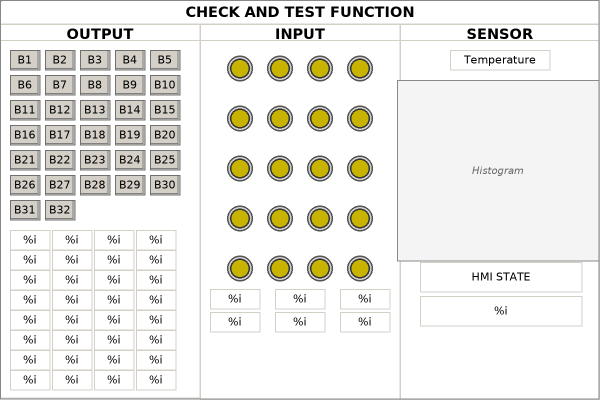
VISUALIZATION Set  // 600x400
    Textfield (0,0 600x24), "CHECK AND TEST FUNCTION"
    Rectangle (0,0 1x0)
    Textfield (0,24 200x20), "OUTPUT"
    Textfield (200,24 200x20), "INPUT"
    Textfield (400,24 200x20), "SENSOR"
    Textfield (0,40 200x358)
    Textfield (200,40 200x360)
    Textfield (400,40 200x360)
    Lamp1 (225,51 30x35), variable: HMI_Global.HMI_IN_Digital[0], style: Lamp-Lamp1-Yellow
    Lamp1 (265,51 30x35), variable: HMI_Global.HMI_IN_Digital[1], style: Lamp-Lamp1-Yellow
    Lamp1 (305,51 30x35), variable: HMI_Global.HMI_IN_Digital[2], style: Lamp-Lamp1-Yellow
    Lamp1 (345,51 30x35), variable: HMI_Global.HMI_IN_Digital[3], style: Lamp-Lamp1-Yellow
    Lamp1 (345,101 30x35), variable: HMI_Global.HMI_IN_Digital[7], style: Lamp-Lamp1-Yellow
    Lamp1 (225,101 30x35), variable: HMI_Global.HMI_IN_Digital[4], style: Lamp-Lamp1-Yellow
    Lamp1 (265,101 30x35), variable: HMI_Global.HMI_IN_Digital[5], style: Lamp-Lamp1-Yellow
    Lamp1 (305,101 30x35), variable: HMI_Global.HMI_IN_Digital[6], style: Lamp-Lamp1-Yellow
    Lamp1 (225,151 30x35), variable: HMI_Global.HMI_IN_Digital[8], style: Lamp-Lamp1-Yellow
    Lamp1 (345,151 30x35), variable: HMI_Global.HMI_IN_Digital[11], style: Lamp-Lamp1-Yellow
    Lamp1 (265,151 30x35), variable: HMI_Global.HMI_IN_Digital[9], style: Lamp-Lamp1-Yellow
    Lamp1 (305,151 30x35), variable: HMI_Global.HMI_IN_Digital[10], style: Lamp-Lamp1-Yellow
    Lamp1 (225,201 30x35), variable: HMI_Global.HMI_IN_Digital[12], style: Lamp-Lamp1-Yellow
    Lamp1 (265,201 30x35), variable: HMI_Global.HMI_IN_Digital[13], style: Lamp-Lamp1-Yellow
    Lamp1 (305,201 30x35), variable: HMI_Global.HMI_IN_Digital[14], style: Lamp-Lamp1-Yellow
    Lamp1 (345,201 30x35), variable: HMI_Global.HMI_IN_Digital[15], style: Lamp-Lamp1-Yellow
    Lamp1 (345,251 30x35), variable: HMI_Global.HMI_IN_Digital[20], style: Lamp-Lamp1-Yellow
    Lamp1 (225,251 30x35), variable: HMI_Global.HMI_IN_Digital[16], style: Lamp-Lamp1-Yellow
    Lamp1 (265,251 30x35), variable: HMI_Global.HMI_IN_Digital[17], style: Lamp-Lamp1-Yellow
    Lamp1 (305,251 30x35), variable: HMI_Global.HMI_IN_Digital[18], style: Lamp-Lamp1-Yellow
    Button (10,50 30x20), "B1"
        toggle HMI_Global.HMI_OUT_Digital[0]
    Textfield (210,289 50x20), "%i", text variable: HMI_Global.HMI_IN_Analog[0]
    Textfield (275,289 50x20), "%i", text variable: HMI_Global.HMI_IN_Analog[1]
    Textfield (340,289 50x20), "%i", text variable: HMI_Global.HMI_IN_Analog[2]
    Textfield (210,312 50x20), "%i", text variable: HMI_Global.HMI_IN_Analog[3]
    Textfield (275,312 50x20), "%i", text variable: HMI_Global.HMI_IN_Analog[4]
    Textfield (340,312 50x20), "%i", text variable: HMI_Global.HMI_IN_Analog[5]
    Textfield (10,230 40x20), "%i", text variable: HMI_Global.HMI_OUT_Analog[0]
        OnMouseDown: write the text variable via VisuDialogs.Numpad, min 0, max 1000
    Histogram (397,80 202x181), scale format: %.1f, scale 0..100
        p1518820177: HMI_Global.HMI_IN_Temp
        p102497268: HMI_Global.HMI_IN_Temp
        p788070771: ARRAY [0..4] OF REAL
    Textfield (450,50 100x20), "Temperature"
    Textfield (420,262 162x30), "HMI STATE"
    Textfield (420,296 162x30), "%i", text variable: HMI_Global.HMI_State
    Button (45,50 30x20), "B2"
        toggle HMI_Global.HMI_OUT_Digital[1]
    Button (80,50 30x20), "B3"
        toggle HMI_Global.HMI_OUT_Digital[2]
    Button (115,50 30x20), "B4"
        toggle HMI_Global.HMI_OUT_Digital[3]
    Button (150,50 30x20), "B5"
        toggle HMI_Global.HMI_OUT_Digital[4]
    Button (10,75 30x20), "B6"
        toggle HMI_Global.HMI_OUT_Digital[5]
    Button (45,75 30x20), "B7"
        toggle HMI_Global.HMI_OUT_Digital[6]
    Button (80,75 30x20), "B8"
        toggle HMI_Global.HMI_OUT_Digital[7]
    Button (115,75 30x20), "B9"
        toggle HMI_Global.HMI_OUT_Digital[8]
    Button (150,75 30x20), "B10"
        toggle HMI_Global.HMI_OUT_Digital[9]
    Button (10,125 30x20), "B16"
        toggle HMI_Global.HMI_OUT_Digital[15]
    Button (10,100 30x20), "B11"
        toggle HMI_Global.HMI_OUT_Digital[10]
    Button (45,100 30x20), "B12"
        toggle HMI_Global.HMI_OUT_Digital[11]
    Button (80,100 30x20), "B13"
        toggle HMI_Global.HMI_OUT_Digital[12]
    Button (115,100 30x20), "B14"
        toggle HMI_Global.HMI_OUT_Digital[13]
    Button (150,100 30x20), "B15"
        toggle HMI_Global.HMI_OUT_Digital[14]
    Button (45,125 30x20), "B17"
        toggle HMI_Global.HMI_OUT_Digital[16]
    Button (80,125 30x20), "B18"
        toggle HMI_Global.HMI_OUT_Digital[17]
    Button (115,125 30x20), "B19"
        toggle HMI_Global.HMI_OUT_Digital[18]
    Button (150,125 30x20), "B20"
        toggle HMI_Global.HMI_OUT_Digital[19]
    Button (10,150 30x20), "B21"
        toggle HMI_Global.HMI_OUT_Digital[20]
    Button (10,175 30x20), "B26"
        toggle HMI_Global.HMI_OUT_Digital[25]
    Button (45,150 30x20), "B22"
        toggle HMI_Global.HMI_OUT_Digital[21]
    Button (80,150 30x20), "B23"
        toggle HMI_Global.HMI_OUT_Digital[22]
    Button (115,150 30x20), "B24"
        toggle HMI_Global.HMI_OUT_Digital[23]
    Button (150,150 30x20), "B25"
        toggle HMI_Global.HMI_OUT_Digital[24]
    Button (45,175 30x20), "B27"
        toggle HMI_Global.HMI_OUT_Digital[26]
    Button (80,175 30x20), "B28"
        toggle HMI_Global.HMI_OUT_Digital[27]
    Button (115,175 30x20), "B29"
        toggle HMI_Global.HMI_OUT_Digital[28]
    Button (150,175 30x20), "B30"
        toggle HMI_Global.HMI_OUT_Digital[29]
    Button (10,200 30x20), "B31"
        toggle HMI_Global.HMI_OUT_Digital[30]
    Button (45,200 30x20), "B32"
        toggle HMI_Global.HMI_OUT_Digital[31]
    Textfield (52,230 40x20), "%i", text variable: HMI_Global.HMI_OUT_Analog[1]
        OnMouseDown: write the text variable via VisuDialogs.Numpad, min 0, max 1000
    Textfield (94,230 40x20), "%i", text variable: HMI_Global.HMI_OUT_Analog[2]
        OnMouseDown: write the text variable via VisuDialogs.Numpad, min 0, max 1000
    Textfield (136,230 40x20), "%i", text variable: HMI_Global.HMI_OUT_Analog[3]
        OnMouseDown: write the text variable via VisuDialogs.Numpad, min 0, max 1000
    Textfield (10,250 40x20), "%i", text variable: HMI_Global.HMI_OUT_Analog[4]
        OnMouseDown: write the text variable via VisuDialogs.Numpad, min 0, max 1000
    Textfield (52,250 40x20), "%i", text variable: HMI_Global.HMI_OUT_Analog[5]
        OnMouseDown: write the text variable via VisuDialogs.Numpad, min 0, max 1000
    Textfield (94,250 40x20), "%i", text variable: HMI_Global.HMI_OUT_Analog[6]
        OnMouseDown: write the text variable via VisuDialogs.Numpad, min 0, max 1000
    Textfield (136,250 40x20), "%i", text variable: HMI_Global.HMI_OUT_Analog[7]
        OnMouseDown: write the text variable via VisuDialogs.Numpad, min 0, max 1000
    Textfield (10,270 40x20), "%i", text variable: HMI_Global.HMI_OUT_Analog[8]
        OnMouseDown: write the text variable via VisuDialogs.Numpad, min 0, max 1000
    Textfield (52,270 40x20), "%i", text variable: HMI_Global.HMI_OUT_Analog[9]
        OnMouseDown: write the text variable via VisuDialogs.Numpad, min 0, max 1000
    Textfield (94,270 40x20), "%i", text variable: HMI_Global.HMI_OUT_Analog[10]
        OnMouseDown: write the text variable via VisuDialogs.Numpad, min 0, max 1000
    Textfield (136,270 40x20), "%i", text variable: HMI_Global.HMI_OUT_Analog[11]
        OnMouseDown: write the text variable via VisuDialogs.Numpad, min 0, max 1000
    Textfield (10,290 40x20), "%i", text variable: HMI_Global.HMI_OUT_Analog[12]
        OnMouseDown: write the text variable via VisuDialogs.Numpad, min 0, max 1000
    Textfield (52,290 40x20), "%i", text variable: HMI_Global.HMI_OUT_Analog[13]
        OnMouseDown: write the text variable via VisuDialogs.Numpad, min 0, max 1000
    Textfield (94,290 40x20), "%i", text variable: HMI_Global.HMI_OUT_Analog[14]
        OnMouseDown: write the text variable via VisuDialogs.Numpad, min 0, max 1000
    Textfield (136,290 40x20), "%i", text variable: HMI_Global.HMI_OUT_Analog[15]
        OnMouseDown: write the text variable via VisuDialogs.Numpad, min 0, max 1000
    Textfield (10,310 40x20), "%i", text variable: HMI_Global.HMI_OUT_Analog[16]
        OnMouseDown: write the text variable via VisuDialogs.Numpad, min 0, max 1000
    Textfield (52,310 40x20), "%i", text variable: HMI_Global.HMI_OUT_Analog[17]
        OnMouseDown: write the text variable via VisuDialogs.Numpad, min 0, max 1000
    Textfield (94,310 40x20), "%i", text variable: HMI_Global.HMI_OUT_Analog[18]
        OnMouseDown: write the text variable via VisuDialogs.Numpad, min 0, max 1000
    Textfield (136,310 40x20), "%i", text variable: HMI_Global.HMI_OUT_Analog[19]
        OnMouseDown: write the text variable via VisuDialogs.Numpad, min 0, max 1000
    Textfield (10,330 40x20), "%i", text variable: HMI_Global.HMI_OUT_Analog[20]
        OnMouseDown: write the text variable via VisuDialogs.Numpad, min 0, max 1000
    Textfield (52,330 40x20), "%i", text variable: HMI_Global.HMI_OUT_Analog[21]
        OnMouseDown: write the text variable via VisuDialogs.Numpad, min 0, max 1000
    Textfield (94,330 40x20), "%i", text variable: HMI_Global.HMI_OUT_Analog[22]
        OnMouseDown: write the text variable via VisuDialogs.Numpad, min 0, max 1000
    Textfield (136,330 40x20), "%i", text variable: HMI_Global.HMI_OUT_Analog[23]
        OnMouseDown: write the text variable via VisuDialogs.Numpad, min 0, max 1000
    Textfield (10,350 40x20), "%i", text variable: HMI_Global.HMI_OUT_Analog[24]
        OnMouseDown: write the text variable via VisuDialogs.Numpad, min 0, max 1000
    Textfield (52,350 40x20), "%i", text variable: HMI_Global.HMI_OUT_Analog[25]
        OnMouseDown: write the text variable via VisuDialogs.Numpad, min 0, max 1000
    Textfield (94,350 40x20), "%i", text variable: HMI_Global.HMI_OUT_Analog[26]
        OnMouseDown: write the text variable via VisuDialogs.Numpad, min 0, max 1000
    Textfield (136,350 40x20), "%i", text variable: HMI_Global.HMI_OUT_Analog[27]
        OnMouseDown: write the text variable via VisuDialogs.Numpad, min 0, max 1000
    Textfield (10,370 40x20), "%i", text variable: HMI_Global.HMI_OUT_Analog[28]
        OnMouseDown: write the text variable via VisuDialogs.Numpad, min 0, max 1000
    Textfield (52,370 40x20), "%i", text variable: HMI_Global.HMI_OUT_Analog[29]
        OnMouseDown: write the text variable via VisuDialogs.Numpad, min 0, max 1000
    Textfield (94,370 40x20), "%i", text variable: HMI_Global.HMI_OUT_Analog[30]
        OnMouseDown: write the text variable via VisuDialogs.Numpad, min 0, max 1000
    Textfield (136,370 40x20), "%i", text variable: HMI_Global.HMI_OUT_Analog[31]
        OnMouseDown: write the text variable via VisuDialogs.Numpad, min 0, max 1000
END_VISUALIZATION

(* stored: Version 1.1.0.1, ProductVersion 3.1.4024.12
   Visu Set: Id {c9cc3fe0-fd97-4ebc-826a-4a84b7032f61} *)
